FUNCTION IsGreaterThanOrEqualAnyType : E_GeneralResult
VAR_INPUT
	A					: __SYSTEM.AnyType; // A and B have to be same type
	B					: __SYSTEM.AnyType; // A and B have to be same type
END_VAR

IsGreaterThanOrEqualAnyType := NegateGeneralResult(IsLessThanAnyType(A, B));

END_FUNCTION

(* stored: Version 1.1.0.1, ProductVersion 3.1.4024.11
   POU IsGreaterThanOrEqualAnyType: Id {de59629a-5382-42b5-8401-14196fcf1f98}, SpecialFunc None *)
